FUNCTION_BLOCK FB_Crossing
VAR_INPUT
	bCDayMode : BOOL;
	stMainIn : ST_TrafficLightInput;
	stSubIn : ST_TrafficLightInput;
END_VAR
VAR_OUTPUT
END_VAR
VAR
	fbTrafficLightArray : ARRAY[1..4] OF FB_TrafficLight; //defining the array
	idx : INT;
	tonCrossing : TON;
	nStep : INT;
	
END_VAR


CASE nStep OF
	
	0:  IF NOT bCDayMode THEN
			stMainIn.bDayMode := FALSE;
			stSubIn.bDayMode := FALSE;
		ELSE 
			stMainIn.bDayMode := TRUE;
			stSubIn.bDayMode := TRUE;
			nStep := 10;
		END_IF
	10: stMainIn.bSetRed := TRUE;
		stSubIn.bSetRed := TRUE;
		tonCrossing(IN := TRUE, PT := T#3S);
		IF tonCrossing.Q AND bCDayMode THEN
			stMainIn.bSetRed := FALSE;
			stSubIn.bSetRed := FALSE;
			tonCrossing(IN := FALSE);
			nStep := 20;
		END_IF
		IF NOT bCDayMode THEN
			tonCrossing(IN := FALSE);
			stMainIn.bSetGreen := TRUE;
			stMainIn.bSetRed := FALSE;
			stSubIn.bSetGreen := TRUE;
			stSubIn.bSetRed := FALSE;
			nStep := 0;
		END_IF
	20: stSubIn.bSetRed := TRUE;
		IF fbTrafficLightArray[3].stTrafficLightOutput.bRed THEN
			stMainIn.bSetGreen := TRUE;
		END_IF
		tonCrossing(IN := TRUE, PT := T#10S);
		IF tonCrossing.Q AND bCDayMode THEN
			tonCrossing(IN := FALSE);
			stMainIn.bSetGreen := FALSE;
			stSubIn.bSetRed := FALSE;
			nStep := 30;
		END_IF
		IF NOT bCDayMode THEN
			tonCrossing(IN := FALSE);
			stMainIn.bSetGreen := FALSE;
			stSubIn.bSetGreen := FALSE;
			nStep := 0;
		END_IF
	30: stMainIn.bSetRed := TRUE;
		IF fbTrafficLightArray[1].stTrafficLightOutput.bRed THEN
			stSubIn.bSetGreen := TRUE;
		END_IF
		tonCrossing(IN := TRUE, PT := T#10S);
		IF tonCrossing.Q AND bCDayMode THEN
			tonCrossing(IN := FALSE);
			stMainIn.bSetRed := FALSE;
			stSubIn.bSetGreen := FALSE;
			nStep := 20;
		END_IF
		IF NOT bCDayMode THEN
			tonCrossing(IN := FALSE);
			stMainIn.bSetGreen := FALSE;
			stSubIn.bSetGreen := FALSE;
			nStep := 0;
		END_IF
			
	
END_CASE

FOR idx := 1 TO 2 DO    
			fbTrafficLightArray[idx](stTrafficLightInput := stMainIn);
END_FOR
FOR idx := 3 TO 4 DO    
			fbTrafficLightArray[idx](stTrafficLightInput := stSubIn);
END_FOR

END_FUNCTION_BLOCK

(* stored: Version 1.1.0.1, ProductVersion 3.1.4024.0
   POU FB_Crossing: Id {7f7f13c2-ef31-4491-9dde-30a8b67eee87}, SpecialFunc None *)
